{region '#Template'}
	{attribute 'Category' := 'DUTs'}
	{attribute 'Version' := '0.0.1.0'}
	{attribute 'Tags' := 'Operation mode, Universal, Modulation'}
	{attribute 'Description' := 'Modulationsbefehle // modulation commands'}
{endregion}
{attribute 'qualified_only'}
TYPE E_BA_MdltCmd :
(
	eOff			:= 1,
	eOn				:= 2,
	eMin			:= 3,
	eMax			:= 4
	
) UDINT;
END_TYPE

(* stored: Version 1.1.0.1, ProductVersion 3.1.4024.6
   DUT E_BA_MdltCmd: Id {2b7380a6-e66f-4c3c-932a-6a2d900ab432} *)
